FUNCTION AddToArray : BOOL
VAR_INPUT
	arr : POINTER TO BYTE;
	numEntries : LINT;
	dataSize : UDINT;
	
	newEntry : ANY;
END_VAR
VAR
	i : LINT;
END_VAR

//numEntries := (UPPER_BOUND(arr, 1) - LOWER_BOUND(arr, 1) + 1) / dataSize;

FOR i:=0 TO numEntries-1 BY 1 DO
	
	IF ArrayIsEmpty(arr := ADR(arr[i]), arrSize := dataSize) THEN
		AddToArray := MEMCPY(ADR(arr[i]), ADR(newEntry), dataSize) > 0;
		RETURN;
	END_IF
	
END_FOR

END_FUNCTION

(* stored: Version 1.1.0.1, ProductVersion 3.1.4024.11
   POU AddToArray: Id {e5ab1016-66e7-4d55-91ab-7f206e04401d}, SpecialFunc None *)
